PROGRAM System_1
VAR

	
	Always_ON					:	BOOL	:=TRUE;	//상시ON
	Always_OFF					:	BOOL	:=FALSE;//상시OFF

	TON_ON  					: 	TON		; 		// 0.1초 ON 타이머 인스턴스
    TON_OFF 					:	TON		; 		// 0.1초 OFF 타이머 인스턴스
	TON2_ON  					: 	TON		; 		// 1초 ON 타이머 인스턴스
    TON2_OFF 					:	TON		;		 // 1초 OFF 타이머 인스턴스
	
	IO_Test						:	BOOL	;
	Lamp_Test_Green				:	BOOL	;
	Lamp_Test_Yellow			:	BOOL	;
	Lamp_Test_Red				:	BOOL	;
	Lamp_Test_Buzzer			:	BOOL	;
	Moving_Motor_Wait_Position: BOOL;
END_VAR
VAR // added by the converter: edge detectors and wires of the graphical bodies
    _rt1, _rt2, _rt3, _rt4, _rt5, _rt6 : R_TRIG;
END_VAR

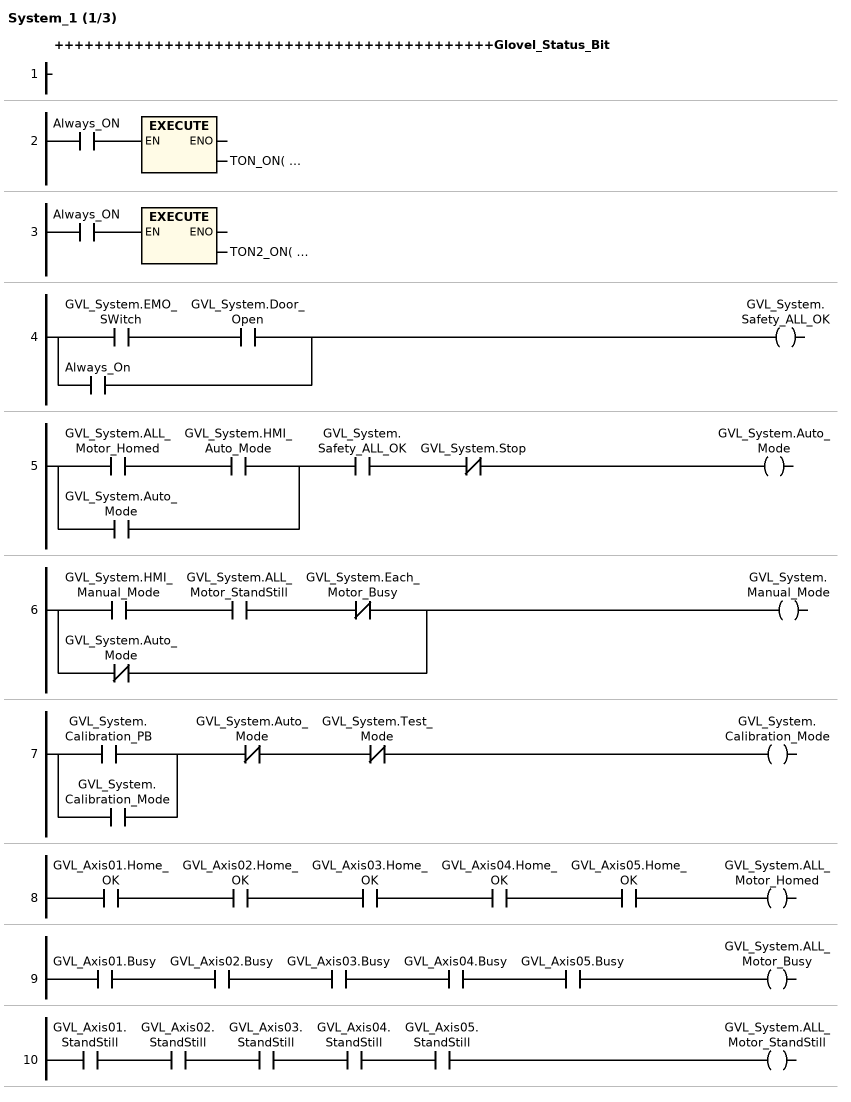
// NETWORK 1: ++++++++++++++++++++++++++++++++++++++++++++Glovel_Status_Bit

// NETWORK 2
IF Always_ON THEN
    TON_ON(
        IN := Always_ON AND NOT TON_OFF.Q,
        PT := T#100ms,
        Q  => 
    );
    
    TON_OFF(
        IN := Always_ON AND TON_ON.Q, 
        PT := T#100ms,
        Q  => 
    );
    
    GVL_System.Pulse_100ms := TON_OFF.IN;
END_IF

// NETWORK 3
IF Always_ON THEN
    TON2_ON(
        IN := Always_ON AND NOT TON2_OFF.Q,
        PT := T#1S,
        Q  => 
    );
    
    TON2_OFF(
        IN := Always_ON AND TON2_ON.Q,
        PT := T#1S,
        Q  => 
    );
    
    GVL_System.Pulse_1S := TON2_OFF.IN;
END_IF

// NETWORK 4
GVL_System.Safety_ALL_OK := GVL_System.EMO_SWitch AND GVL_System.Door_Open OR Always_On;

// NETWORK 5
GVL_System.Auto_Mode := (GVL_System.ALL_Motor_Homed AND GVL_System.HMI_Auto_Mode OR GVL_System.Auto_Mode) AND GVL_System.Safety_ALL_OK AND NOT GVL_System.Stop;

// NETWORK 6
GVL_System.Manual_Mode := GVL_System.HMI_Manual_Mode AND GVL_System.ALL_Motor_StandStill AND NOT GVL_System.Each_Motor_Busy OR NOT GVL_System.Auto_Mode;

// NETWORK 7
GVL_System.Calibration_Mode := (GVL_System.Calibration_PB OR GVL_System.Calibration_Mode) AND NOT GVL_System.Auto_Mode AND NOT GVL_System.Test_Mode;

// NETWORK 8
GVL_System.ALL_Motor_Homed := GVL_Axis01.Home_OK AND GVL_Axis02.Home_OK AND GVL_Axis03.Home_OK AND GVL_Axis04.Home_OK AND GVL_Axis05.Home_OK;

// NETWORK 9
GVL_System.ALL_Motor_Busy := GVL_Axis01.Busy AND GVL_Axis02.Busy AND GVL_Axis03.Busy AND GVL_Axis04.Busy AND GVL_Axis05.Busy;

// NETWORK 10
GVL_System.ALL_Motor_StandStill := GVL_Axis01.StandStill AND GVL_Axis02.StandStill AND GVL_Axis03.StandStill AND GVL_Axis04.StandStill AND GVL_Axis05.StandStill;

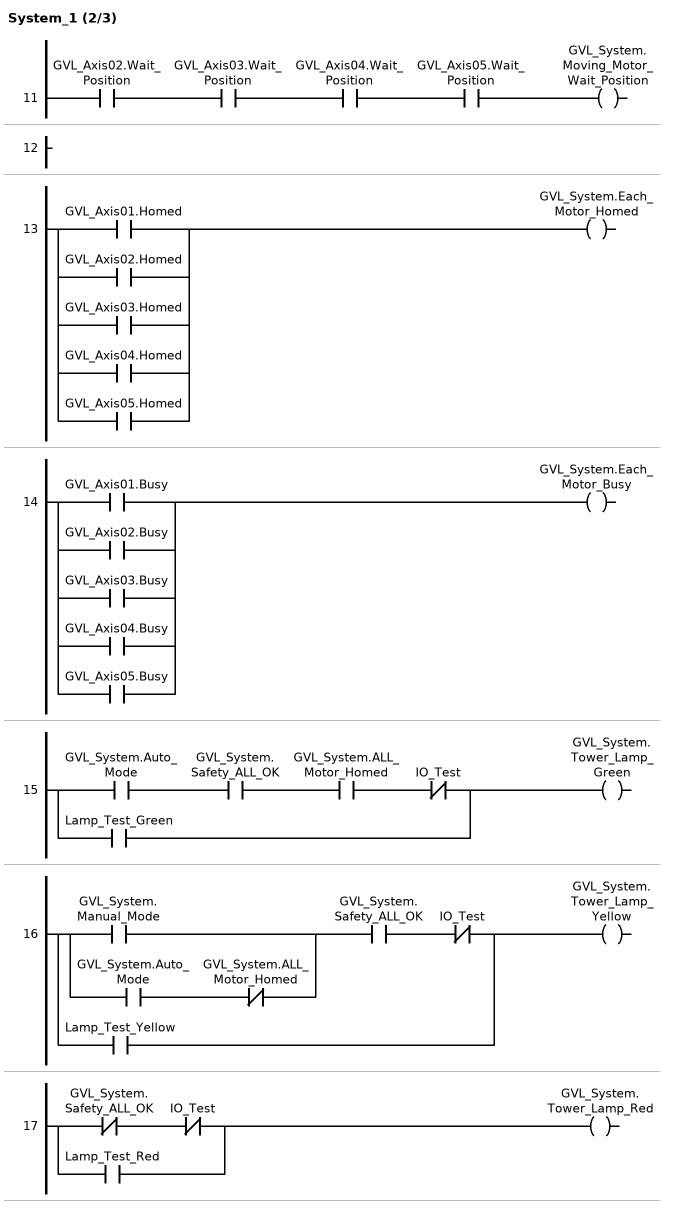
// NETWORK 11
GVL_System.Moving_Motor_Wait_Position := GVL_Axis02.Wait_Position AND GVL_Axis03.Wait_Position AND GVL_Axis04.Wait_Position AND GVL_Axis05.Wait_Position;

// NETWORK 12

// NETWORK 13
GVL_System.Each_Motor_Homed := GVL_Axis01.Homed OR GVL_Axis02.Homed OR GVL_Axis03.Homed OR GVL_Axis04.Homed OR GVL_Axis05.Homed;

// NETWORK 14
GVL_System.Each_Motor_Busy := GVL_Axis01.Busy OR GVL_Axis02.Busy OR GVL_Axis03.Busy OR GVL_Axis04.Busy OR GVL_Axis05.Busy;

// NETWORK 15
GVL_System.Tower_Lamp_Green := GVL_System.Auto_Mode AND GVL_System.Safety_ALL_OK AND GVL_System.ALL_Motor_Homed AND NOT IO_Test OR Lamp_Test_Green;

// NETWORK 16
GVL_System.Tower_Lamp_Yellow := (GVL_System.Manual_Mode OR GVL_System.Auto_Mode AND NOT GVL_System.ALL_Motor_Homed) AND GVL_System.Safety_ALL_OK AND NOT IO_Test OR Lamp_Test_Yellow;

// NETWORK 17
GVL_System.Tower_Lamp_Red := NOT GVL_System.Safety_ALL_OK AND NOT IO_Test OR Lamp_Test_Red;

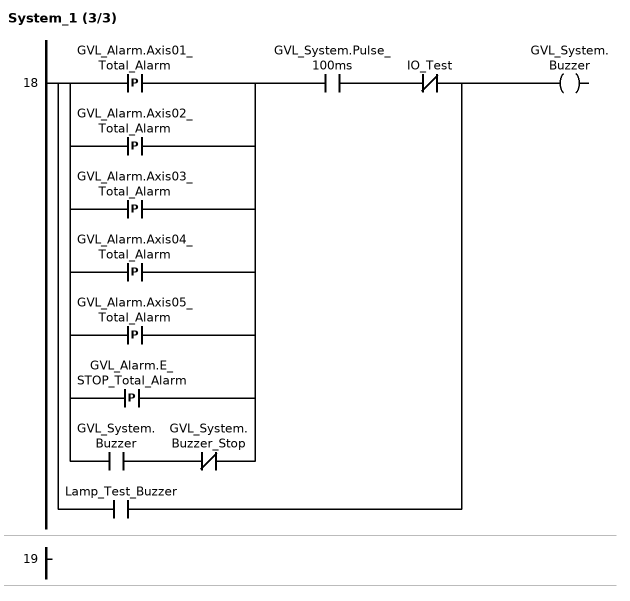
// NETWORK 18
_rt1(CLK := GVL_Alarm.Axis01_Total_Alarm);
_rt2(CLK := GVL_Alarm.Axis02_Total_Alarm);
_rt3(CLK := GVL_Alarm.Axis03_Total_Alarm);
_rt4(CLK := GVL_Alarm.Axis04_Total_Alarm);
_rt5(CLK := GVL_Alarm.Axis05_Total_Alarm);
_rt6(CLK := GVL_Alarm.E_STOP_Total_Alarm);
GVL_System.Buzzer := (_rt1.Q OR _rt2.Q OR _rt3.Q OR _rt4.Q OR _rt5.Q OR _rt6.Q OR GVL_System.Buzzer AND NOT GVL_System.Buzzer_Stop) AND GVL_System.Pulse_100ms AND NOT IO_Test OR Lamp_Test_Buzzer;

// NETWORK 19

END_PROGRAM

(* stored: Version 1.1.0.1, ProductVersion 3.1.4024.15
   POU System_1: Id {79af5364-68b1-49b6-9473-e37ca620de11}, SpecialFunc None *)
